// TIA Portal V18 export
DATA_BLOCK "SS1_A5_16DI_DI_Vars"   // DB11051
{ S7_Optimized_Access := 'FALSE' }
VERSION : 0.1
// stored: AutoNumber false, DBAccessibleFromOPCUA true, IsOnlyStoredInLoadMemory false, IsWriteProtectedInAS false
   VAR
      DI1 : "UDT_DIadv";
      DI2 : "UDT_DIadv";
      DI3 : "UDT_DIadv";
      DI4 : "UDT_DIadv";
      DI5 : "UDT_DIadv";
      DI6 : "UDT_DIadv";
      DI7 : "UDT_DIadv";
      DI8 : "UDT_DIadv";
      DI9 { S7_SetPoint := 'True'} : "UDT_DIadv";
      DI10 { S7_SetPoint := 'True'} : "UDT_DIadv";
      DI11 { S7_SetPoint := 'True'} : "UDT_DIadv";
      DI12 { S7_SetPoint := 'True'} : "UDT_DIadv";
      DI13 { S7_SetPoint := 'True'} : "UDT_DIadv";
      DI14 { S7_SetPoint := 'True'} : "UDT_DIadv";
      DI15 { S7_SetPoint := 'True'} : "UDT_DIadv";
      DI16 { S7_SetPoint := 'True'} : "UDT_DIadv";
   END_VAR
BEGIN
   DI3.cFuncSystemID := 10;
   DI3.cFuncVar := 25;
   DI4.cFuncSystemID := 10;
   DI4.cFuncVar := 26;
   DI5.cFuncSystemID := 10;
   DI5.cFuncVar := 27;
   DI6.cFuncSystemID := 100;
   DI6.cFuncVar := 11;
   DI7.cFuncSystemID := 100;
   DI7.cFuncVar := 12;
   DI8.cFuncSystemID := 10;
   DI8.cFuncVar := 24;
   DI9.cFuncSystemID := 10;
   DI9.cFuncVar := 22;
   DI10.xInversion := true;
   DI10.cFuncSystemID := 10;
   DI10.cFuncVar := 23;
   DI11.cFuncSystemID := 10;
   DI11.cFuncVar := 7;
   DI12.cFuncSystemID := 10;
   DI12.cFuncVar := 2;
   DI13.xInversion := true;
   DI13.cFuncSystemID := 10;
   DI13.cFuncVar := 3;
   DI14.cFuncSystemID := 10;
   DI14.cFuncVar := 5;
   DI15.xInversion := true;
   DI15.cFuncSystemID := 10;
   DI15.cFuncVar := 6;
END_DATA_BLOCK
